Omron CX-Programmer project NewProject (CX-Programmer 9.81)

# PLC Sessao_07_04_2026_Exercicio: CP1L M
; 

## Global symbols (name address type ; comment)
0.00 BOOL  ; Botao Start
0.01 BOOL  ; Botao Start 1
0.02 BOOL  ; Botao Reset
0.03 BOOL  ; Botao Stop
0.04 BOOL  ; Botao Start
0.05 BOOL  ; Botao Start 1
0.06 BOOL  ; Botao de Emergencia 2
0.07 BOOL  ; Botao Stop 1
0.08 BOOL  ; Flag do Temporizador 1
0.09 BOOL  ; Botao de Start Esquerdo
0.10 BOOL  ; Botao de Start Direito
0.11 BOOL  ; Temporizador
100 CHANNEL  ; Temporizador
100.00 BOOL  ; Pulso
100.01 BOOL  ; Actuador
100.02 BOOL  ; Motor Garra
100.03 BOOL  ; Pulso 1
100.04 BOOL  ; Actuador 1
100.05 BOOL  ; Contactor
100.06 BOOL  ; Bobina do Motor 2
100.07 BOOL  ; Temporizador
2.00 BOOL  ; Actuador
4 CHANNEL  ; Contador
500 CHANNEL  ; Temporizador 1
C0004 BOOL  ; Contador
T0001 BOOL  ; Flag do Temporizador 1

## Program NewProgram1 (cyclic task 0)
Local symbols
A 100.02 BOOL  ; Actuador
B_Start 0.00 BOOL  ; Botao Start
P 100.01 BOOL  ; Pulso
R 100.00 BOOL  ; Botao Reset

### Section Exercicio_1_Pulso

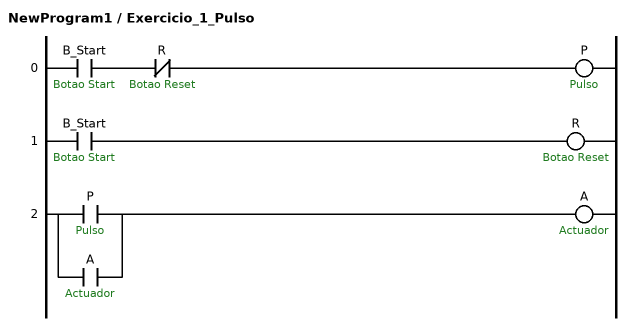
; rung 0
LD B_Start  ; Botao Start
ANDNOT R  ; Botao Reset
OUT P  ; Pulso
; rung 1
LD B_Start  ; Botao Start
OUT R  ; Botao Reset
; rung 2
LD P  ; Pulso
OR A  ; Actuador
OUT A  ; Actuador

### Section END
; rung 0
END(001)